Staubli VAL3: FINDSTR.pgx

public program FindStr(string x_sFindStr, string& x_sStrArray[], num& x_nPos)
  local num l_nSize
  local num i
begin
  //在x_sStrArray中查找x_sFindStr
  //x_nPos:位置
  //
  l_nSize=size(x_sStrArray)
  for  i=0 to l_nSize-1
    if x_sFindStr==x_sStrArray[i]
      x_nPos=i
      return
    endIf
  endFor
  x_nPos=-1
end
